Fanuc KAREL source: kb00071.KL

-- PROVISIONAL review KL for V940-1; original PC SHA256 d8170aabfc80a6809f0c46043e31b3812b805b7c10ac64df0a49dc57e1d8280d
-- Incomplete behavior may be omitted. Consult companion uncertainty JSON. Do not deploy.
PROGRAM KB00071
%NOLOCKGROUP
VAR
  P1 : REAL
  RESULT : REAL
BEGIN
  -- V9_ZERO_TABLE_METADATA_HINT layout=0001; no indexed target words; source/name/runtime held
  -- UNRESOLVED_PC offsets 5-16; opcodes 2E,23
  -- UNRESOLVED_PC offsets 21-36; opcodes 27,22,76,23
  -- UNRESOLVED_PC offsets 41-45; opcodes 7F
END KB00071
